FUNCTION_BLOCK LogMessage IMPLEMENTS I_LogMessage
VAR
	{attribute 'hide'}
	_Message : T_MaxString;
	{attribute 'hide'}
	_Severity : USINT;
END_VAR

{attribute 'monitoring':='call'}
PROPERTY Message : T_MaxString
GET
Message := _Message;
END_GET
SET
_Message := Message;
END_SET
END_PROPERTY

{attribute 'monitoring':='call'}
PROPERTY Severity : USINT
GET
Severity := _Severity;
END_GET
SET
_Severity := Severity;
END_SET
END_PROPERTY

END_FUNCTION_BLOCK

(* stored: Version 1.1.0.1, ProductVersion 3.1.4026.18
   POU LogMessage: Id {6744a647-59d8-4a0e-b6fa-34f9ee18a173}, SpecialFunc None
   Property Message: Id {e9f13044-6913-4c1e-89ff-e281fe3caeec}
   Get Get: Id {c9aa7f3f-bd9d-4ea0-b4f7-926d1a9d54d8}
   Set Set: Id {e61b5359-3e1b-4418-a3b3-35230b74f67e}
   Property Severity: Id {dc09d0d2-da80-42d1-afc3-835a9cd678f6}
   Get Get: Id {ac033b73-5da9-4d83-8f50-3528599b4d83}
   Set Set: Id {cf1b165f-7e93-478e-8d08-5a14c026c9af} *)
